// Startup hook called before Init and PostInit.
INTERFACE I_PreInit EXTENDS I_Generic

// Called once during Plant startup before Init.
METHOD PreInit
END_METHOD

END_INTERFACE

(* stored: Version 1.1.0.1
   Itf I_PreInit: Id {86558393-4550-4676-9af0-3feafb797384}
   Method PreInit: Id {4a3a1e05-aa4f-4dba-965f-466f8ae16c7e} *)
